(* PLC project Unnamed, Неизвестно Unnamed 1 *)
(* stored: creationDateTime 2024-03-29T11:42:58, modificationDateTime 2024-03-29T17:55:06 *)

PROGRAM PWM
  VAR
    duty_fb AT %QW2 : WORD;
    freq AT %QW1 : WORD;
  END_VAR
  VAR
    freq_real : REAL;
  END_VAR
  VAR
    duty AT %QW0 : WORD;
  END_VAR
  VAR
    PWM_CONTROLLER0 : PWM_CONTROLLER;
  END_VAR

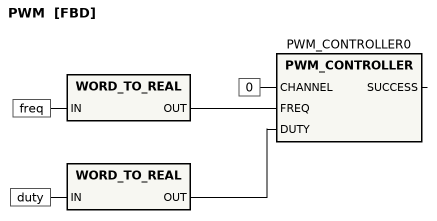
(* FBD diagram, written out as Structured Text *)
PWM_CONTROLLER0(CHANNEL := 0, FREQ := WORD_TO_REAL(freq), DUTY := WORD_TO_REAL(duty));
END_PROGRAM

CONFIGURATION Config0
  RESOURCE Res0 ON PLC
    TASK task0(INTERVAL := T#20ms, PRIORITY := 0);
    PROGRAM instance0 WITH task0 : PWM;
  END_RESOURCE
END_CONFIGURATION
